(* CoDeSys 2.3.9.50 project: 5E.pr6 *)
(* Libraries: STANDARD.LB6 5.6.98 12:03:02 *)

(* POU MAIN, LD *)
PROGRAM MAIN
VAR
	Start AT %IX0.0: BOOL;
	Conveyer1count AT %IX0.1: BOOL;
	Conveyer2count AT %IX0.2: BOOL;
	Conveyer3count AT %IX0.3: BOOL;
	C1: CTU;
	C2: CTU;
	C3: CTU;
	Reset AT %IX0.7: BOOL;
	T1: TON;

	Total: INT;
END_VAR
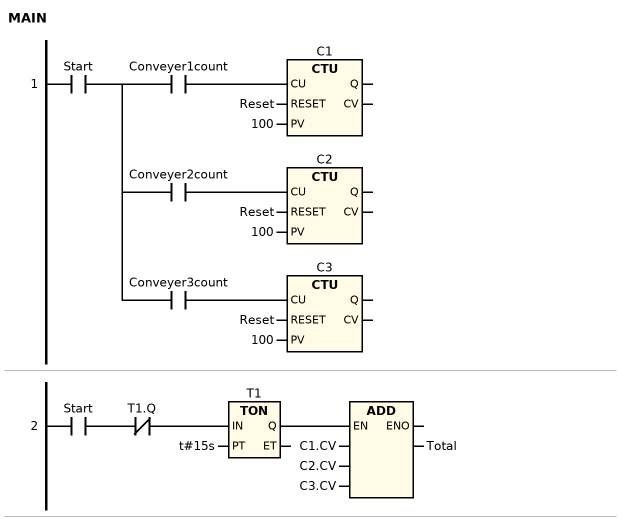
_LD_ (* Ladder Diagram *)
NETWORK 1
	[Start] - { [Conveyer1count] - C1:CTU(CU: *, RESET: Reset, PV: 100) | [Conveyer2count] - C2:CTU(CU: *, RESET: Reset, PV: 100) | [Conveyer3count] - C3:CTU(CU: *, RESET: Reset, PV: 100) }
NETWORK 2
	[Start] - [/T1.Q] - T1:TON(IN: *, PT: t#15s)
		EN --- ADD(C1.CV, C2.CV, C3.CV) => Total
_END_LD_
(* the same logic as Structured Text *)
(* Network 1 *)
C1(CU := Start AND Conveyer1count, RESET := Reset, PV := 100);
C2(CU := Start AND Conveyer2count, RESET := Reset, PV := 100);
C3(CU := Start AND Conveyer3count, RESET := Reset, PV := 100);
(* Network 2 *)
T1(IN := Start AND NOT T1.Q, PT := t#15s);
IF T1.Q THEN
	Total := C1.CV + C2.CV + C3.CV;
END_IF;
END_PROGRAM
